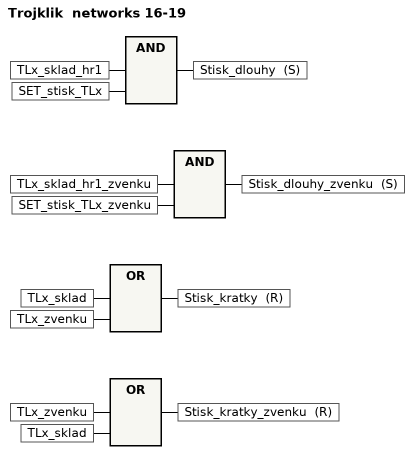
[picture p24: Trojklik (FBD) networks 16-19]
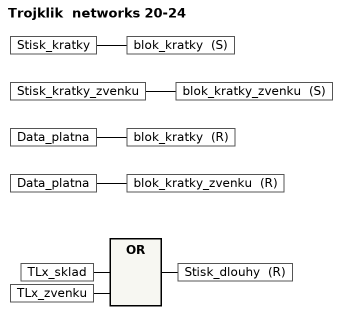
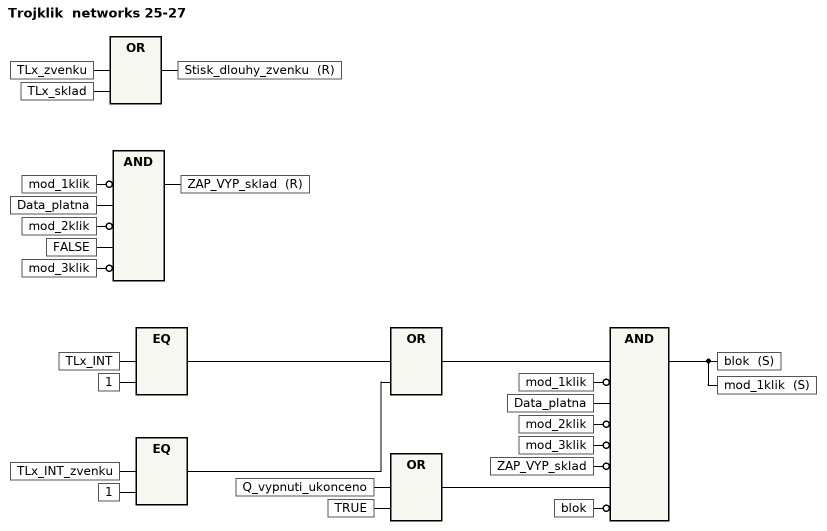
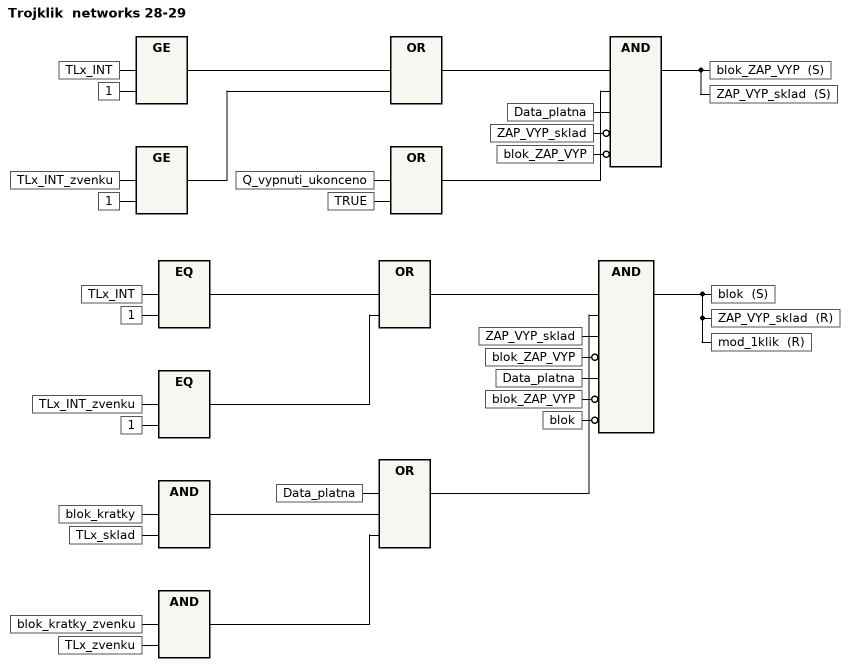
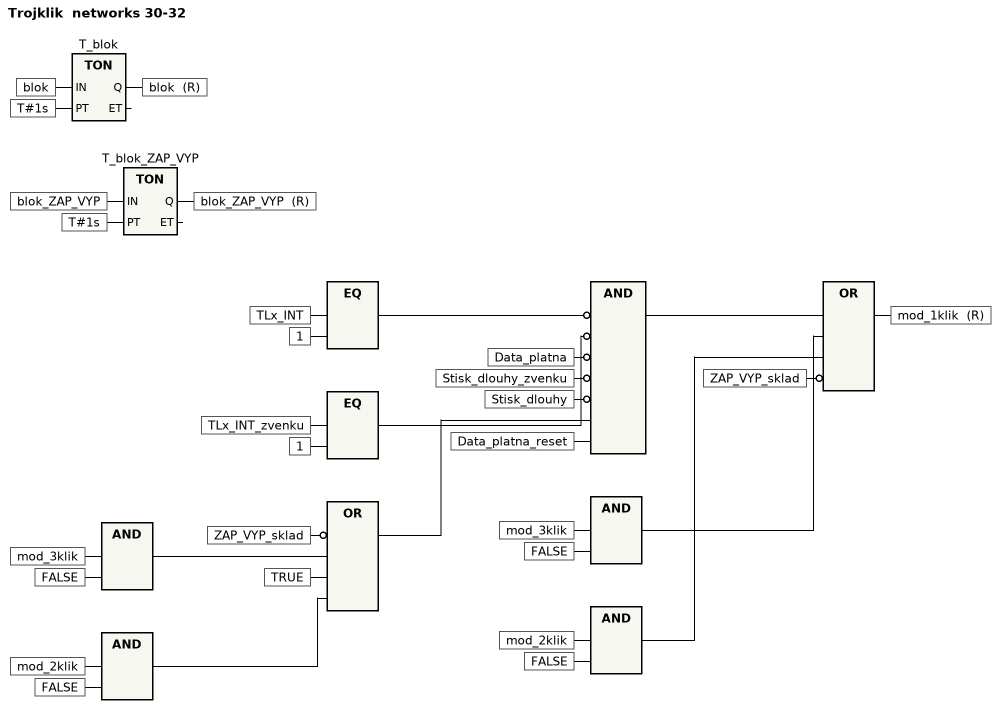
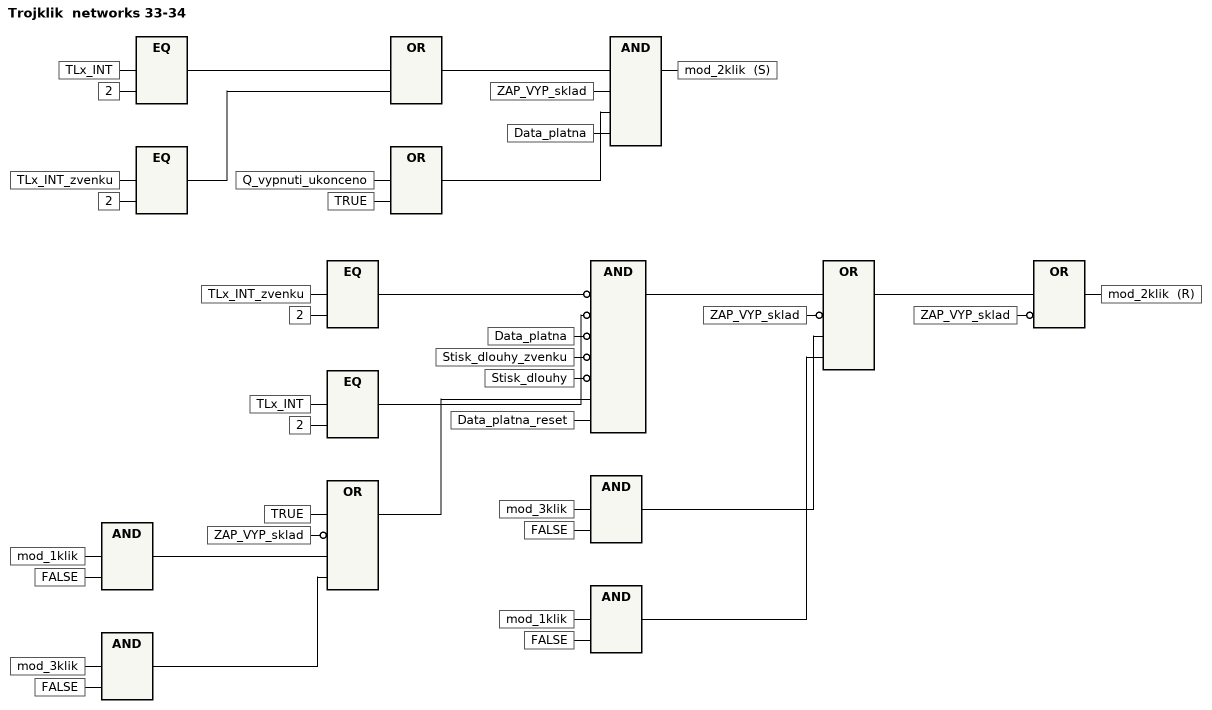
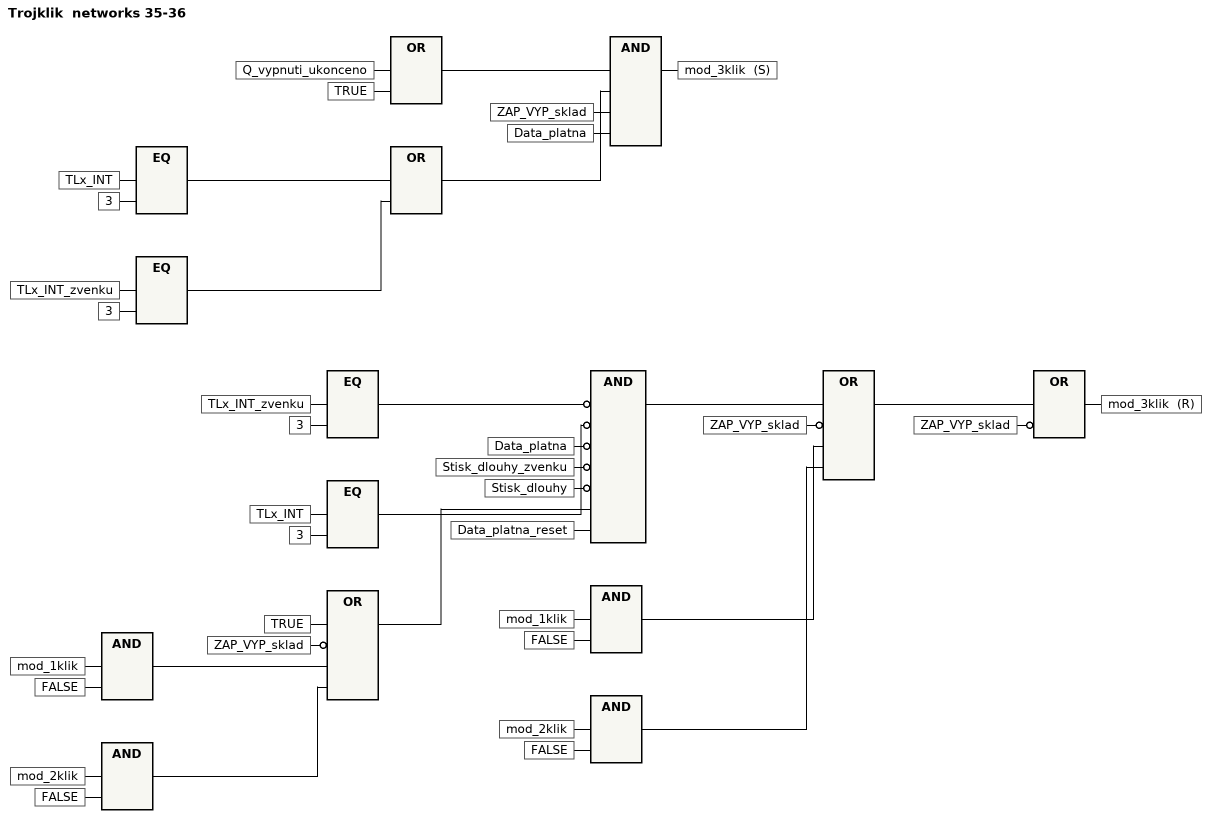
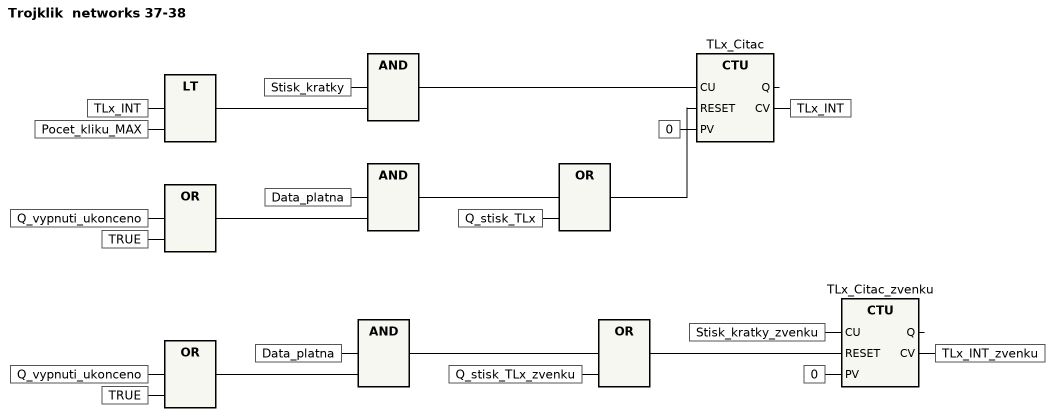
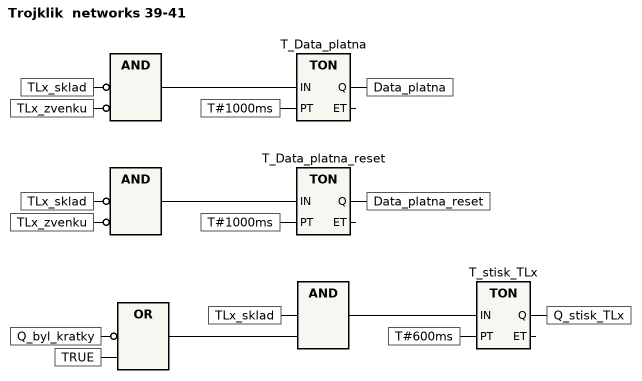
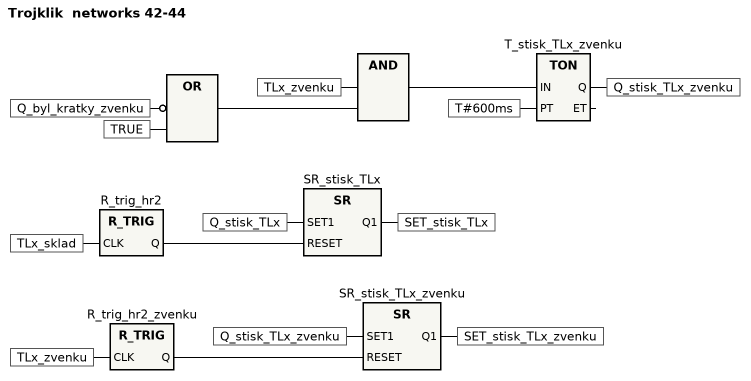
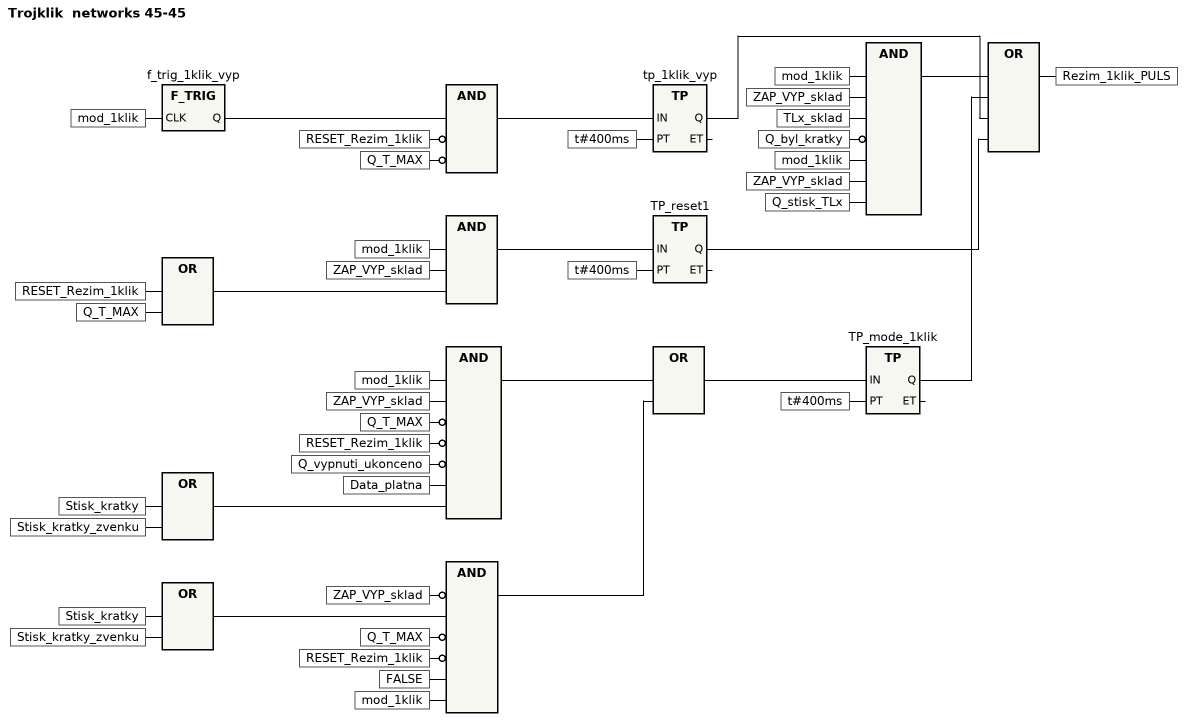
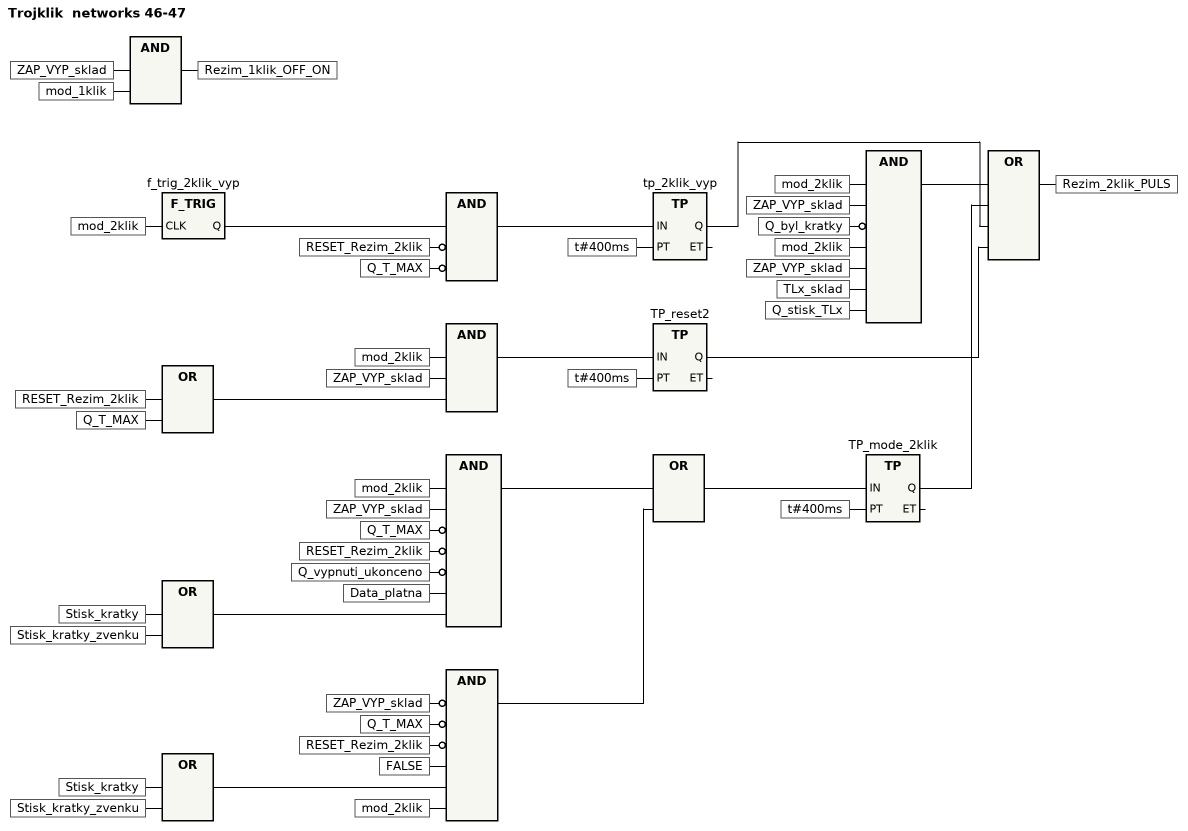
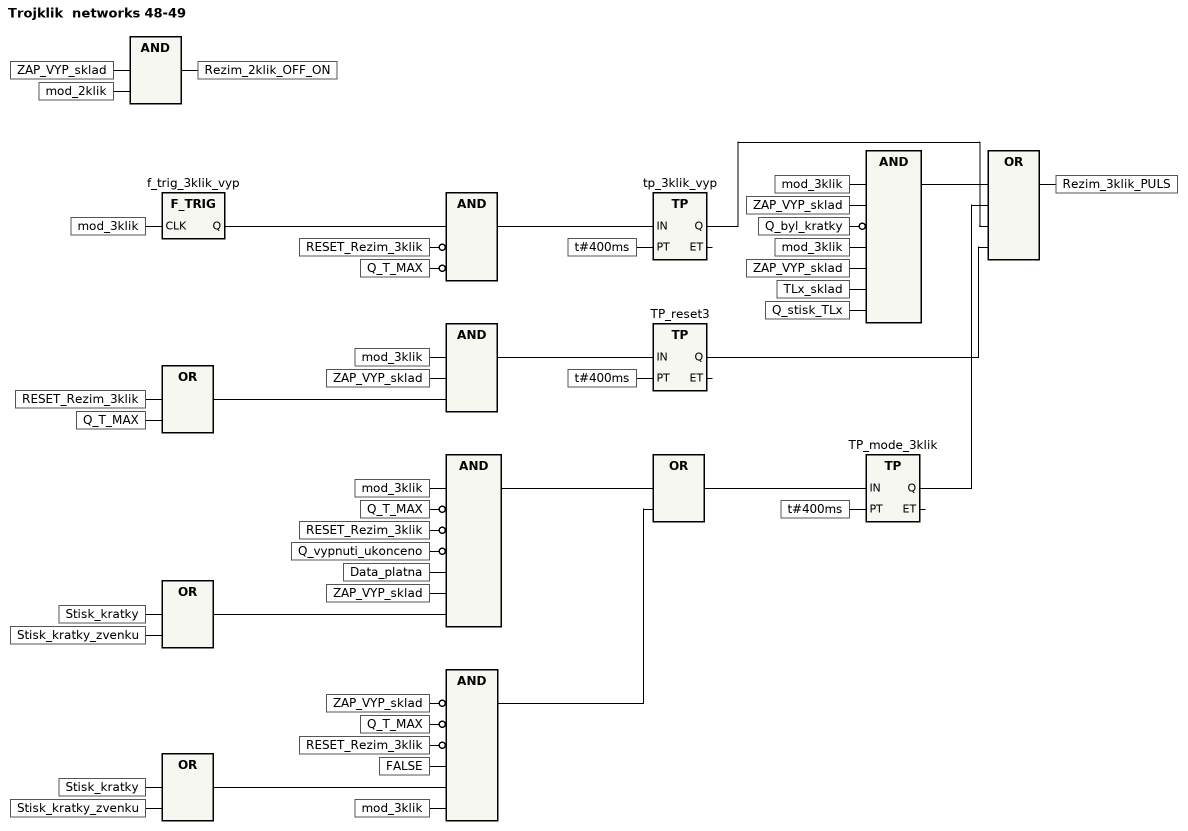
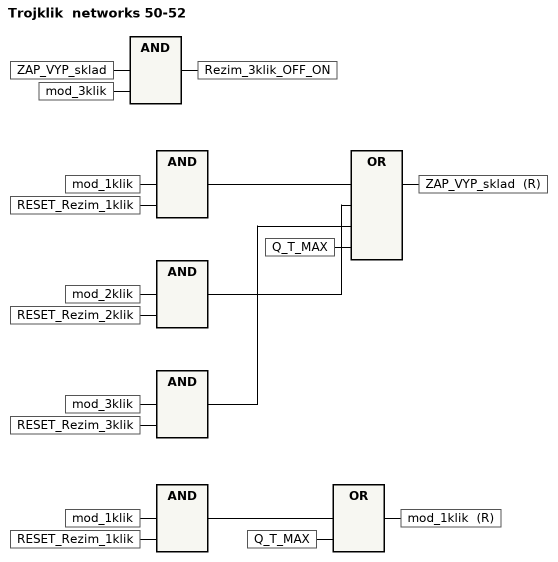
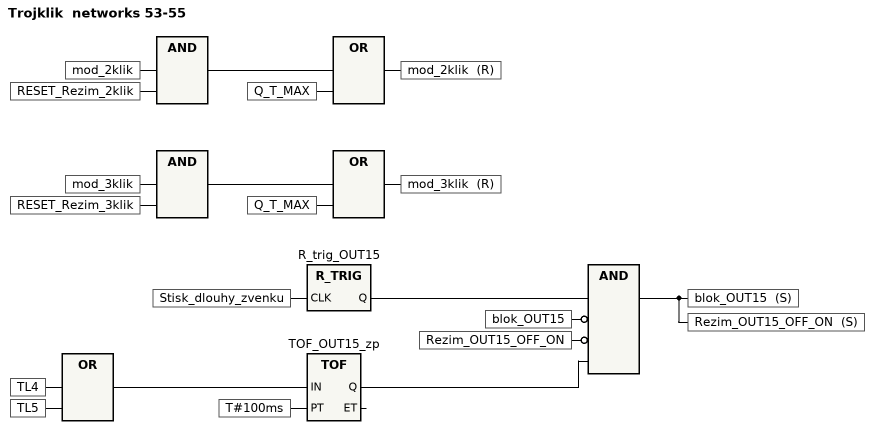
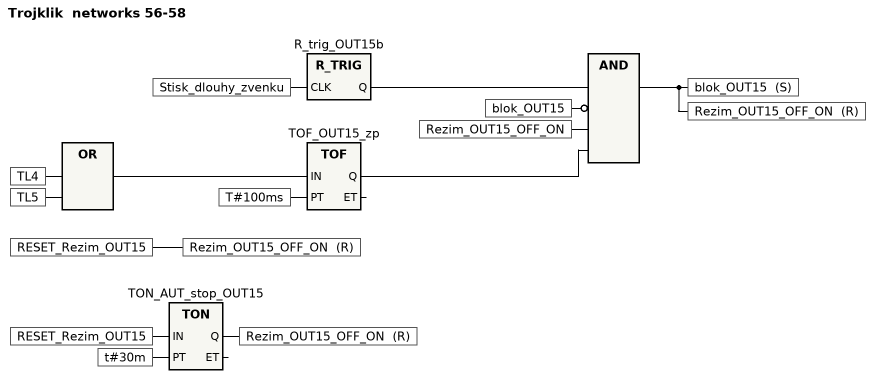
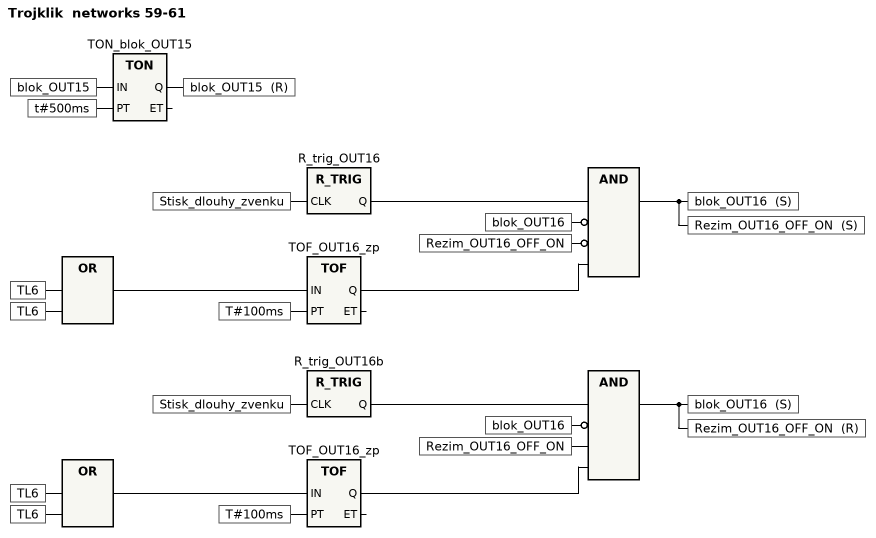
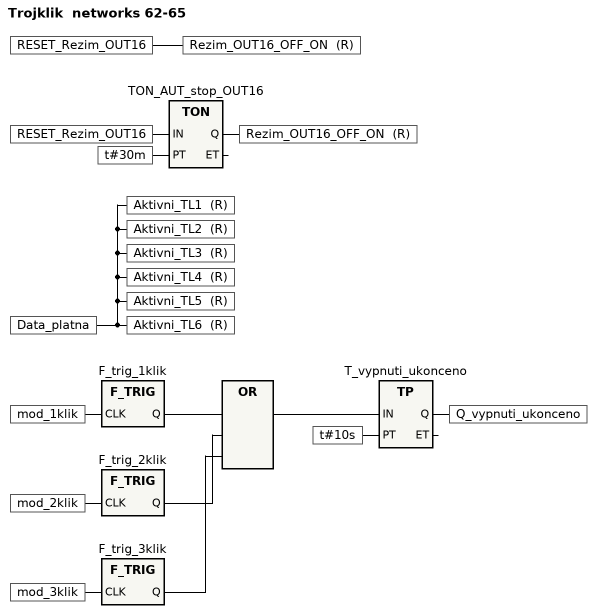
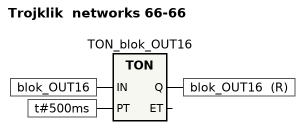
_FBD_ (* Function Block Diagram *)
NETWORK 1
	TP_T_max:TP(IN: T_max:TON(IN: AND(OR(Rezim_1klik_OFF_ON, Rezim_2klik_OFF_ON, Rezim_3klik_OFF_ON), AUT_vyp), PT: cas_vypnuti), PT: t#400ms) => Q_T_MAX
NETWORK 2
	AND(TL1, NOT Aktivni_TL1, NOT Aktivni_TL2, NOT Aktivni_TL3, NOT Aktivni_TL4, NOT Aktivni_TL5, NOT Aktivni_TL6) => S Aktivni_TL1
NETWORK 3
	AND(TL2, NOT Aktivni_TL1, NOT Aktivni_TL2, NOT Aktivni_TL3, NOT Aktivni_TL4, NOT Aktivni_TL5, NOT Aktivni_TL6) => S Aktivni_TL2
NETWORK 4
	AND(TL3, NOT Aktivni_TL1, NOT Aktivni_TL2, NOT Aktivni_TL3, NOT Aktivni_TL4, NOT Aktivni_TL5, NOT Aktivni_TL6) => S Aktivni_TL3
NETWORK 5
	AND(TL4, NOT Aktivni_TL1, NOT Aktivni_TL2, NOT Aktivni_TL3, NOT Aktivni_TL4, NOT Aktivni_TL5, NOT Aktivni_TL6) => S Aktivni_TL4
NETWORK 6
	AND(TL5, NOT Aktivni_TL1, NOT Aktivni_TL2, NOT Aktivni_TL3, NOT Aktivni_TL4, NOT Aktivni_TL5, NOT Aktivni_TL6) => S Aktivni_TL5
NETWORK 7
	AND(TL6, NOT Aktivni_TL1, NOT Aktivni_TL2, NOT Aktivni_TL3, NOT Aktivni_TL4, NOT Aktivni_TL5, NOT Aktivni_TL6) => S Aktivni_TL6
NETWORK 8
	OR(AND(TL1, Aktivni_TL1), AND(TL2, Aktivni_TL2), AND(TL3, Aktivni_TL3)) => TLx_sklad
NETWORK 9
	OR(AND(TL4, Aktivni_TL4), AND(TL5, Aktivni_TL5), AND(TL6, Aktivni_TL6)) => TLx_zvenku
NETWORK 10
	F_trig_hr1:F_TRIG(CLK: TLx_sklad) => TLx_sklad_hr1
NETWORK 11
	F_trig_hr1_zvenku:F_TRIG(CLK: TLx_zvenku) => TLx_sklad_hr1_zvenku
NETWORK 12
	AND(TLx_sklad_hr1, NOT SET_stisk_TLx) => S Stisk_kratky
NETWORK 13
	AND(TLx_sklad_hr1_zvenku, NOT SET_stisk_TLx_zvenku) => S Stisk_kratky_zvenku
NETWORK 14
	TP_byl_kratky:TP(IN: Stisk_kratky, PT: T#4s) => Q_byl_kratky
NETWORK 15
	TP_byl_kratky_zvenku:TP(IN: Stisk_kratky_zvenku, PT: T#4s) => Q_byl_kratky_zvenku
NETWORK 16
	AND(TLx_sklad_hr1, SET_stisk_TLx) => S Stisk_dlouhy
NETWORK 17
	AND(TLx_sklad_hr1_zvenku, SET_stisk_TLx_zvenku) => S Stisk_dlouhy_zvenku
NETWORK 18
	OR(TLx_sklad, TLx_zvenku) => R Stisk_kratky
NETWORK 19
	OR(TLx_zvenku, TLx_sklad) => R Stisk_kratky_zvenku
NETWORK 20
	Stisk_kratky => S blok_kratky
NETWORK 21
	Stisk_kratky_zvenku => S blok_kratky_zvenku
NETWORK 22
	Data_platna => R blok_kratky
NETWORK 23
	Data_platna => R blok_kratky_zvenku
NETWORK 24
	OR(TLx_sklad, TLx_zvenku) => R Stisk_dlouhy
NETWORK 25
	OR(TLx_zvenku, TLx_sklad) => R Stisk_dlouhy_zvenku
NETWORK 26
	AND(NOT mod_1klik, Data_platna, NOT mod_2klik, FALSE, NOT mod_3klik) => R ZAP_VYP_sklad
NETWORK 27
	AND(OR(EQ(TLx_INT, 1), EQ(TLx_INT_zvenku, 1)), NOT mod_1klik, Data_platna, NOT mod_2klik, NOT mod_3klik, NOT ZAP_VYP_sklad, OR(Q_vypnuti_ukonceno, TRUE), NOT blok) => S blok, S mod_1klik
NETWORK 28
	AND(OR(GE(TLx_INT, 1), GE(TLx_INT_zvenku, 1)), OR(Q_vypnuti_ukonceno, TRUE), Data_platna, NOT ZAP_VYP_sklad, NOT blok_ZAP_VYP) => S blok_ZAP_VYP, S ZAP_VYP_sklad
NETWORK 29
	AND(OR(EQ(TLx_INT, 1), EQ(TLx_INT_zvenku, 1)), OR(Data_platna, AND(blok_kratky, TLx_sklad), AND(blok_kratky_zvenku, TLx_zvenku)), ZAP_VYP_sklad, NOT blok_ZAP_VYP, Data_platna, NOT blok_ZAP_VYP, NOT blok) => S blok, R ZAP_VYP_sklad, R mod_1klik
NETWORK 30
	T_blok:TON(IN: blok, PT: T#1s) => R blok
NETWORK 31
	T_blok_ZAP_VYP:TON(IN: blok_ZAP_VYP, PT: T#1s) => R blok_ZAP_VYP
NETWORK 32
	OR(AND(NOT EQ(TLx_INT, 1), NOT EQ(TLx_INT_zvenku, 1), NOT Data_platna, NOT Stisk_dlouhy_zvenku, NOT Stisk_dlouhy, OR(NOT ZAP_VYP_sklad, AND(mod_3klik, FALSE), TRUE, AND(mod_2klik, FALSE)), Data_platna_reset), AND(mod_3klik, FALSE), AND(mod_2klik, FALSE), NOT ZAP_VYP_sklad) => R mod_1klik
NETWORK 33
	AND(OR(EQ(TLx_INT, 2), EQ(TLx_INT_zvenku, 2)), ZAP_VYP_sklad, OR(Q_vypnuti_ukonceno, TRUE), Data_platna) => S mod_2klik
NETWORK 34
	OR(OR(AND(NOT EQ(TLx_INT_zvenku, 2), NOT EQ(TLx_INT, 2), NOT Data_platna, NOT Stisk_dlouhy_zvenku, NOT Stisk_dlouhy, OR(TRUE, NOT ZAP_VYP_sklad, AND(mod_1klik, FALSE), AND(mod_3klik, FALSE)), Data_platna_reset), NOT ZAP_VYP_sklad, AND(mod_3klik, FALSE), AND(mod_1klik, FALSE)), NOT ZAP_VYP_sklad) => R mod_2klik
NETWORK 35
	AND(OR(Q_vypnuti_ukonceno, TRUE), OR(EQ(TLx_INT, 3), EQ(TLx_INT_zvenku, 3)), ZAP_VYP_sklad, Data_platna) => S mod_3klik
NETWORK 36
	OR(OR(AND(NOT EQ(TLx_INT_zvenku, 3), NOT EQ(TLx_INT, 3), NOT Data_platna, NOT Stisk_dlouhy_zvenku, NOT Stisk_dlouhy, OR(TRUE, NOT ZAP_VYP_sklad, AND(mod_1klik, FALSE), AND(mod_2klik, FALSE)), Data_platna_reset), NOT ZAP_VYP_sklad, AND(mod_1klik, FALSE), AND(mod_2klik, FALSE)), NOT ZAP_VYP_sklad) => R mod_3klik
NETWORK 37
	TLx_Citac:CTU(CU: AND(Stisk_kratky, LT(TLx_INT, Pocet_kliku_MAX)), RESET: OR(AND(Data_platna, OR(Q_vypnuti_ukonceno, TRUE)), Q_stisk_TLx), PV: 0, CV => TLx_INT)
NETWORK 38
	TLx_Citac_zvenku:CTU(CU: Stisk_kratky_zvenku, RESET: OR(AND(Data_platna, OR(Q_vypnuti_ukonceno, TRUE)), Q_stisk_TLx_zvenku), PV: 0, CV => TLx_INT_zvenku)
NETWORK 39 (* Data platna *)
	T_Data_platna:TON(IN: AND(NOT TLx_sklad, NOT TLx_zvenku), PT: T#1000ms) => Data_platna
NETWORK 40 (* Data platna *)
	T_Data_platna_reset:TON(IN: AND(NOT TLx_sklad, NOT TLx_zvenku), PT: T#1000ms) => Data_platna_reset
NETWORK 41 (* delka stisku TLx *)
	T_stisk_TLx:TON(IN: AND(TLx_sklad, OR(NOT Q_byl_kratky, TRUE)), PT: T#600ms) => Q_stisk_TLx
NETWORK 42 (* delka stisku TLx *)
	T_stisk_TLx_zvenku:TON(IN: AND(TLx_zvenku, OR(NOT Q_byl_kratky_zvenku, TRUE)), PT: T#600ms) => Q_stisk_TLx_zvenku
NETWORK 43
	SR_stisk_TLx:SR(SET1: Q_stisk_TLx, RESET: R_trig_hr2:R_TRIG(CLK: TLx_sklad)) => SET_stisk_TLx
NETWORK 44
	SR_stisk_TLx_zvenku:SR(SET1: Q_stisk_TLx_zvenku, RESET: R_trig_hr2_zvenku:R_TRIG(CLK: TLx_zvenku)) => SET_stisk_TLx_zvenku
NETWORK 45
	OR(AND(mod_1klik, ZAP_VYP_sklad, TLx_sklad, NOT Q_byl_kratky, mod_1klik, ZAP_VYP_sklad, Q_stisk_TLx), TP_mode_1klik:TP(IN: OR(AND(mod_1klik, ZAP_VYP_sklad, NOT Q_T_MAX, NOT RESET_Rezim_1klik, NOT Q_vypnuti_ukonceno, Data_platna, OR(Stisk_kratky, Stisk_kratky_zvenku)), AND(NOT ZAP_VYP_sklad, OR(Stisk_kratky, Stisk_kratky_zvenku), NOT Q_T_MAX, NOT RESET_Rezim_1klik, FALSE, mod_1klik)), PT: t#400ms), tp_1klik_vyp:TP(IN: AND(f_trig_1klik_vyp:F_TRIG(CLK: mod_1klik), NOT RESET_Rezim_1klik, NOT Q_T_MAX), PT: t#400ms), TP_reset1:TP(IN: AND(mod_1klik, ZAP_VYP_sklad, OR(RESET_Rezim_1klik, Q_T_MAX)), PT: t#400ms)) => Rezim_1klik_PULS
NETWORK 46
	AND(ZAP_VYP_sklad, mod_1klik) => Rezim_1klik_OFF_ON
NETWORK 47
	OR(AND(mod_2klik, ZAP_VYP_sklad, NOT Q_byl_kratky, mod_2klik, ZAP_VYP_sklad, TLx_sklad, Q_stisk_TLx), TP_mode_2klik:TP(IN: OR(AND(mod_2klik, ZAP_VYP_sklad, NOT Q_T_MAX, NOT RESET_Rezim_2klik, NOT Q_vypnuti_ukonceno, Data_platna, OR(Stisk_kratky, Stisk_kratky_zvenku)), AND(NOT ZAP_VYP_sklad, NOT Q_T_MAX, NOT RESET_Rezim_2klik, FALSE, OR(Stisk_kratky, Stisk_kratky_zvenku), mod_2klik)), PT: t#400ms), tp_2klik_vyp:TP(IN: AND(f_trig_2klik_vyp:F_TRIG(CLK: mod_2klik), NOT RESET_Rezim_2klik, NOT Q_T_MAX), PT: t#400ms), TP_reset2:TP(IN: AND(mod_2klik, ZAP_VYP_sklad, OR(RESET_Rezim_2klik, Q_T_MAX)), PT: t#400ms)) => Rezim_2klik_PULS
NETWORK 48
	AND(ZAP_VYP_sklad, mod_2klik) => Rezim_2klik_OFF_ON
NETWORK 49
	OR(AND(mod_3klik, ZAP_VYP_sklad, NOT Q_byl_kratky, mod_3klik, ZAP_VYP_sklad, TLx_sklad, Q_stisk_TLx), TP_mode_3klik:TP(IN: OR(AND(mod_3klik, NOT Q_T_MAX, NOT RESET_Rezim_3klik, NOT Q_vypnuti_ukonceno, Data_platna, ZAP_VYP_sklad, OR(Stisk_kratky, Stisk_kratky_zvenku)), AND(NOT ZAP_VYP_sklad, NOT Q_T_MAX, NOT RESET_Rezim_3klik, FALSE, OR(Stisk_kratky, Stisk_kratky_zvenku), mod_3klik)), PT: t#400ms), tp_3klik_vyp:TP(IN: AND(f_trig_3klik_vyp:F_TRIG(CLK: mod_3klik), NOT RESET_Rezim_3klik, NOT Q_T_MAX), PT: t#400ms), TP_reset3:TP(IN: AND(mod_3klik, ZAP_VYP_sklad, OR(RESET_Rezim_3klik, Q_T_MAX)), PT: t#400ms)) => Rezim_3klik_PULS
NETWORK 50
	AND(ZAP_VYP_sklad, mod_3klik) => Rezim_3klik_OFF_ON
NETWORK 51
	OR(AND(mod_1klik, RESET_Rezim_1klik), AND(mod_2klik, RESET_Rezim_2klik), AND(mod_3klik, RESET_Rezim_3klik), Q_T_MAX) => R ZAP_VYP_sklad
NETWORK 52
	OR(AND(mod_1klik, RESET_Rezim_1klik), Q_T_MAX) => R mod_1klik
NETWORK 53
	OR(AND(mod_2klik, RESET_Rezim_2klik), Q_T_MAX) => R mod_2klik
NETWORK 54
	OR(AND(mod_3klik, RESET_Rezim_3klik), Q_T_MAX) => R mod_3klik
NETWORK 55
	AND(R_trig_OUT15:R_TRIG(CLK: Stisk_dlouhy_zvenku), NOT blok_OUT15, NOT Rezim_OUT15_OFF_ON, TOF_OUT15_zp:TOF(IN: OR(TL4, TL5), PT: T#100ms)) => S blok_OUT15, S Rezim_OUT15_OFF_ON
NETWORK 56
	AND(R_trig_OUT15b:R_TRIG(CLK: Stisk_dlouhy_zvenku), NOT blok_OUT15, Rezim_OUT15_OFF_ON, TOF_OUT15_zp:TOF(IN: OR(TL4, TL5), PT: T#100ms)) => S blok_OUT15, R Rezim_OUT15_OFF_ON
NETWORK 57
	RESET_Rezim_OUT15 => R Rezim_OUT15_OFF_ON
NETWORK 58
	TON_AUT_stop_OUT15:TON(IN: RESET_Rezim_OUT15, PT: t#30m) => R Rezim_OUT15_OFF_ON
NETWORK 59
	TON_blok_OUT15:TON(IN: blok_OUT15, PT: t#500ms) => R blok_OUT15
NETWORK 60
	AND(R_trig_OUT16:R_TRIG(CLK: Stisk_dlouhy_zvenku), NOT blok_OUT16, NOT Rezim_OUT16_OFF_ON, TOF_OUT16_zp:TOF(IN: OR(TL6, TL6), PT: T#100ms)) => S blok_OUT16, S Rezim_OUT16_OFF_ON
NETWORK 61
	AND(R_trig_OUT16b:R_TRIG(CLK: Stisk_dlouhy_zvenku), NOT blok_OUT16, Rezim_OUT16_OFF_ON, TOF_OUT16_zp:TOF(IN: OR(TL6, TL6), PT: T#100ms)) => S blok_OUT16, R Rezim_OUT16_OFF_ON
NETWORK 62
	RESET_Rezim_OUT16 => R Rezim_OUT16_OFF_ON
NETWORK 63
	TON_AUT_stop_OUT16:TON(IN: RESET_Rezim_OUT16, PT: t#30m) => R Rezim_OUT16_OFF_ON
NETWORK 64
	Data_platna => R Aktivni_TL1, R Aktivni_TL2, R Aktivni_TL3, R Aktivni_TL4, R Aktivni_TL5, R Aktivni_TL6
NETWORK 65
	T_vypnuti_ukonceno:TP(IN: OR(F_trig_1klik:F_TRIG(CLK: mod_1klik), F_trig_2klik:F_TRIG(CLK: mod_2klik), F_trig_3klik:F_TRIG(CLK: mod_3klik)), PT: t#10s) => Q_vypnuti_ukonceno
NETWORK 66
	TON_blok_OUT16:TON(IN: blok_OUT16, PT: t#500ms) => R blok_OUT16
_END_FBD_
(* the same logic as Structured Text *)
(* Network 1 *)
T_max(IN := (Rezim_1klik_OFF_ON OR Rezim_2klik_OFF_ON OR Rezim_3klik_OFF_ON) AND AUT_vyp, PT := cas_vypnuti);
TP_T_max(IN := T_max.Q, PT := t#400ms);
Q_T_MAX := TP_T_max.Q;
(* Network 2 *)
IF TL1 AND NOT Aktivni_TL1 AND NOT Aktivni_TL2 AND NOT Aktivni_TL3 AND NOT Aktivni_TL4 AND NOT Aktivni_TL5 AND NOT Aktivni_TL6 THEN Aktivni_TL1 := TRUE; END_IF;
(* Network 3 *)
IF TL2 AND NOT Aktivni_TL1 AND NOT Aktivni_TL2 AND NOT Aktivni_TL3 AND NOT Aktivni_TL4 AND NOT Aktivni_TL5 AND NOT Aktivni_TL6 THEN Aktivni_TL2 := TRUE; END_IF;
(* Network 4 *)
IF TL3 AND NOT Aktivni_TL1 AND NOT Aktivni_TL2 AND NOT Aktivni_TL3 AND NOT Aktivni_TL4 AND NOT Aktivni_TL5 AND NOT Aktivni_TL6 THEN Aktivni_TL3 := TRUE; END_IF;
(* Network 5 *)
IF TL4 AND NOT Aktivni_TL1 AND NOT Aktivni_TL2 AND NOT Aktivni_TL3 AND NOT Aktivni_TL4 AND NOT Aktivni_TL5 AND NOT Aktivni_TL6 THEN Aktivni_TL4 := TRUE; END_IF;
(* Network 6 *)
IF TL5 AND NOT Aktivni_TL1 AND NOT Aktivni_TL2 AND NOT Aktivni_TL3 AND NOT Aktivni_TL4 AND NOT Aktivni_TL5 AND NOT Aktivni_TL6 THEN Aktivni_TL5 := TRUE; END_IF;
(* Network 7 *)
IF TL6 AND NOT Aktivni_TL1 AND NOT Aktivni_TL2 AND NOT Aktivni_TL3 AND NOT Aktivni_TL4 AND NOT Aktivni_TL5 AND NOT Aktivni_TL6 THEN Aktivni_TL6 := TRUE; END_IF;
(* Network 8 *)
TLx_sklad := (TL1 AND Aktivni_TL1) OR (TL2 AND Aktivni_TL2) OR (TL3 AND Aktivni_TL3);
(* Network 9 *)
TLx_zvenku := (TL4 AND Aktivni_TL4) OR (TL5 AND Aktivni_TL5) OR (TL6 AND Aktivni_TL6);
(* Network 10 *)
F_trig_hr1(CLK := TLx_sklad);
TLx_sklad_hr1 := F_trig_hr1.Q;
(* Network 11 *)
F_trig_hr1_zvenku(CLK := TLx_zvenku);
TLx_sklad_hr1_zvenku := F_trig_hr1_zvenku.Q;
(* Network 12 *)
IF TLx_sklad_hr1 AND NOT SET_stisk_TLx THEN Stisk_kratky := TRUE; END_IF;
(* Network 13 *)
IF TLx_sklad_hr1_zvenku AND NOT SET_stisk_TLx_zvenku THEN Stisk_kratky_zvenku := TRUE; END_IF;
(* Network 14 *)
TP_byl_kratky(IN := Stisk_kratky, PT := T#4s);
Q_byl_kratky := TP_byl_kratky.Q;
(* Network 15 *)
TP_byl_kratky_zvenku(IN := Stisk_kratky_zvenku, PT := T#4s);
Q_byl_kratky_zvenku := TP_byl_kratky_zvenku.Q;
(* Network 16 *)
IF TLx_sklad_hr1 AND SET_stisk_TLx THEN Stisk_dlouhy := TRUE; END_IF;
(* Network 17 *)
IF TLx_sklad_hr1_zvenku AND SET_stisk_TLx_zvenku THEN Stisk_dlouhy_zvenku := TRUE; END_IF;
(* Network 18 *)
IF TLx_sklad OR TLx_zvenku THEN Stisk_kratky := FALSE; END_IF;
(* Network 19 *)
IF TLx_zvenku OR TLx_sklad THEN Stisk_kratky_zvenku := FALSE; END_IF;
(* Network 20 *)
IF Stisk_kratky THEN blok_kratky := TRUE; END_IF;
(* Network 21 *)
IF Stisk_kratky_zvenku THEN blok_kratky_zvenku := TRUE; END_IF;
(* Network 22 *)
IF Data_platna THEN blok_kratky := FALSE; END_IF;
(* Network 23 *)
IF Data_platna THEN blok_kratky_zvenku := FALSE; END_IF;
(* Network 24 *)
IF TLx_sklad OR TLx_zvenku THEN Stisk_dlouhy := FALSE; END_IF;
(* Network 25 *)
IF TLx_zvenku OR TLx_sklad THEN Stisk_dlouhy_zvenku := FALSE; END_IF;
(* Network 26 *)
IF NOT mod_1klik AND Data_platna AND NOT mod_2klik AND FALSE AND NOT mod_3klik THEN ZAP_VYP_sklad := FALSE; END_IF;
(* Network 27 *)
_p1 := ((TLx_INT = 1) OR (TLx_INT_zvenku = 1)) AND NOT mod_1klik AND Data_platna AND NOT mod_2klik AND NOT mod_3klik AND NOT ZAP_VYP_sklad AND (Q_vypnuti_ukonceno OR TRUE) AND NOT blok;
IF _p1 THEN blok := TRUE; mod_1klik := TRUE; END_IF;
(* Network 28 *)
_p2 := ((TLx_INT >= 1) OR (TLx_INT_zvenku >= 1)) AND (Q_vypnuti_ukonceno OR TRUE) AND Data_platna AND NOT ZAP_VYP_sklad AND NOT blok_ZAP_VYP;
IF _p2 THEN blok_ZAP_VYP := TRUE; ZAP_VYP_sklad := TRUE; END_IF;
(* Network 29 *)
_p3 := ((TLx_INT = 1) OR (TLx_INT_zvenku = 1)) AND (Data_platna OR (blok_kratky AND TLx_sklad) OR (blok_kratky_zvenku AND TLx_zvenku)) AND ZAP_VYP_sklad AND NOT blok_ZAP_VYP AND Data_platna AND NOT blok_ZAP_VYP AND NOT blok;
IF _p3 THEN blok := TRUE; ZAP_VYP_sklad := FALSE; mod_1klik := FALSE; END_IF;
(* Network 30 *)
T_blok(IN := blok, PT := T#1s);
IF T_blok.Q THEN blok := FALSE; END_IF;
(* Network 31 *)
T_blok_ZAP_VYP(IN := blok_ZAP_VYP, PT := T#1s);
IF T_blok_ZAP_VYP.Q THEN blok_ZAP_VYP := FALSE; END_IF;
(* Network 32 *)
IF (NOT (TLx_INT = 1) AND NOT (TLx_INT_zvenku = 1) AND NOT Data_platna AND NOT Stisk_dlouhy_zvenku AND NOT Stisk_dlouhy AND (NOT ZAP_VYP_sklad OR (mod_3klik AND FALSE) OR TRUE OR (mod_2klik AND FALSE)) AND Data_platna_reset) OR (mod_3klik AND FALSE) OR (mod_2klik AND FALSE) OR NOT ZAP_VYP_sklad THEN mod_1klik := FALSE; END_IF;
(* Network 33 *)
IF ((TLx_INT = 2) OR (TLx_INT_zvenku = 2)) AND ZAP_VYP_sklad AND (Q_vypnuti_ukonceno OR TRUE) AND Data_platna THEN mod_2klik := TRUE; END_IF;
(* Network 34 *)
IF ((NOT (TLx_INT_zvenku = 2) AND NOT (TLx_INT = 2) AND NOT Data_platna AND NOT Stisk_dlouhy_zvenku AND NOT Stisk_dlouhy AND (TRUE OR NOT ZAP_VYP_sklad OR (mod_1klik AND FALSE) OR (mod_3klik AND FALSE)) AND Data_platna_reset) OR NOT ZAP_VYP_sklad OR (mod_3klik AND FALSE) OR (mod_1klik AND FALSE)) OR NOT ZAP_VYP_sklad THEN mod_2klik := FALSE; END_IF;
(* Network 35 *)
IF (Q_vypnuti_ukonceno OR TRUE) AND ((TLx_INT = 3) OR (TLx_INT_zvenku = 3)) AND ZAP_VYP_sklad AND Data_platna THEN mod_3klik := TRUE; END_IF;
(* Network 36 *)
IF ((NOT (TLx_INT_zvenku = 3) AND NOT (TLx_INT = 3) AND NOT Data_platna AND NOT Stisk_dlouhy_zvenku AND NOT Stisk_dlouhy AND (TRUE OR NOT ZAP_VYP_sklad OR (mod_1klik AND FALSE) OR (mod_2klik AND FALSE)) AND Data_platna_reset) OR NOT ZAP_VYP_sklad OR (mod_1klik AND FALSE) OR (mod_2klik AND FALSE)) OR NOT ZAP_VYP_sklad THEN mod_3klik := FALSE; END_IF;
(* Network 37 *)
TLx_Citac(CU := Stisk_kratky AND (TLx_INT < Pocet_kliku_MAX), RESET := (Data_platna AND (Q_vypnuti_ukonceno OR TRUE)) OR Q_stisk_TLx, PV := 0);
TLx_INT := TLx_Citac.CV;
(* Network 38 *)
TLx_Citac_zvenku(CU := Stisk_kratky_zvenku, RESET := (Data_platna AND (Q_vypnuti_ukonceno OR TRUE)) OR Q_stisk_TLx_zvenku, PV := 0);
TLx_INT_zvenku := TLx_Citac_zvenku.CV;
(* Network 39 *)
T_Data_platna(IN := NOT TLx_sklad AND NOT TLx_zvenku, PT := T#1000ms);
Data_platna := T_Data_platna.Q;
(* Network 40 *)
T_Data_platna_reset(IN := NOT TLx_sklad AND NOT TLx_zvenku, PT := T#1000ms);
Data_platna_reset := T_Data_platna_reset.Q;
(* Network 41: see the listing above *)
(* Network 42: see the listing above *)
(* Network 43 *)
R_trig_hr2(CLK := TLx_sklad);
SR_stisk_TLx(SET1 := Q_stisk_TLx, RESET := R_trig_hr2.Q);
SET_stisk_TLx := SR_stisk_TLx.Q1;
(* Network 44 *)
R_trig_hr2_zvenku(CLK := TLx_zvenku);
SR_stisk_TLx_zvenku(SET1 := Q_stisk_TLx_zvenku, RESET := R_trig_hr2_zvenku.Q);
SET_stisk_TLx_zvenku := SR_stisk_TLx_zvenku.Q1;
(* Network 45 *)
TP_mode_1klik(IN := (mod_1klik AND ZAP_VYP_sklad AND NOT Q_T_MAX AND NOT RESET_Rezim_1klik AND NOT Q_vypnuti_ukonceno AND Data_platna AND (Stisk_kratky OR Stisk_kratky_zvenku)) OR (NOT ZAP_VYP_sklad AND (Stisk_kratky OR Stisk_kratky_zvenku) AND NOT Q_T_MAX AND NOT RESET_Rezim_1klik AND FALSE AND mod_1klik), PT := t#400ms);
f_trig_1klik_vyp(CLK := mod_1klik);
tp_1klik_vyp(IN := f_trig_1klik_vyp.Q AND NOT RESET_Rezim_1klik AND NOT Q_T_MAX, PT := t#400ms);
TP_reset1(IN := mod_1klik AND ZAP_VYP_sklad AND (RESET_Rezim_1klik OR Q_T_MAX), PT := t#400ms);
Rezim_1klik_PULS := (mod_1klik AND ZAP_VYP_sklad AND TLx_sklad AND NOT Q_byl_kratky AND mod_1klik AND ZAP_VYP_sklad AND Q_stisk_TLx) OR TP_mode_1klik.Q OR tp_1klik_vyp.Q OR TP_reset1.Q;
(* Network 46 *)
Rezim_1klik_OFF_ON := ZAP_VYP_sklad AND mod_1klik;
(* Network 47 *)
TP_mode_2klik(IN := (mod_2klik AND ZAP_VYP_sklad AND NOT Q_T_MAX AND NOT RESET_Rezim_2klik AND NOT Q_vypnuti_ukonceno AND Data_platna AND (Stisk_kratky OR Stisk_kratky_zvenku)) OR (NOT ZAP_VYP_sklad AND NOT Q_T_MAX AND NOT RESET_Rezim_2klik AND FALSE AND (Stisk_kratky OR Stisk_kratky_zvenku) AND mod_2klik), PT := t#400ms);
f_trig_2klik_vyp(CLK := mod_2klik);
tp_2klik_vyp(IN := f_trig_2klik_vyp.Q AND NOT RESET_Rezim_2klik AND NOT Q_T_MAX, PT := t#400ms);
TP_reset2(IN := mod_2klik AND ZAP_VYP_sklad AND (RESET_Rezim_2klik OR Q_T_MAX), PT := t#400ms);
Rezim_2klik_PULS := (mod_2klik AND ZAP_VYP_sklad AND NOT Q_byl_kratky AND mod_2klik AND ZAP_VYP_sklad AND TLx_sklad AND Q_stisk_TLx) OR TP_mode_2klik.Q OR tp_2klik_vyp.Q OR TP_reset2.Q;
(* Network 48 *)
Rezim_2klik_OFF_ON := ZAP_VYP_sklad AND mod_2klik;
(* Network 49 *)
TP_mode_3klik(IN := (mod_3klik AND NOT Q_T_MAX AND NOT RESET_Rezim_3klik AND NOT Q_vypnuti_ukonceno AND Data_platna AND ZAP_VYP_sklad AND (Stisk_kratky OR Stisk_kratky_zvenku)) OR (NOT ZAP_VYP_sklad AND NOT Q_T_MAX AND NOT RESET_Rezim_3klik AND FALSE AND (Stisk_kratky OR Stisk_kratky_zvenku) AND mod_3klik), PT := t#400ms);
f_trig_3klik_vyp(CLK := mod_3klik);
tp_3klik_vyp(IN := f_trig_3klik_vyp.Q AND NOT RESET_Rezim_3klik AND NOT Q_T_MAX, PT := t#400ms);
TP_reset3(IN := mod_3klik AND ZAP_VYP_sklad AND (RESET_Rezim_3klik OR Q_T_MAX), PT := t#400ms);
Rezim_3klik_PULS := (mod_3klik AND ZAP_VYP_sklad AND NOT Q_byl_kratky AND mod_3klik AND ZAP_VYP_sklad AND TLx_sklad AND Q_stisk_TLx) OR TP_mode_3klik.Q OR tp_3klik_vyp.Q OR TP_reset3.Q;
(* Network 50 *)
Rezim_3klik_OFF_ON := ZAP_VYP_sklad AND mod_3klik;
(* Network 51 *)
IF (mod_1klik AND RESET_Rezim_1klik) OR (mod_2klik AND RESET_Rezim_2klik) OR (mod_3klik AND RESET_Rezim_3klik) OR Q_T_MAX THEN ZAP_VYP_sklad := FALSE; END_IF;
(* Network 52 *)
IF (mod_1klik AND RESET_Rezim_1klik) OR Q_T_MAX THEN mod_1klik := FALSE; END_IF;
(* Network 53 *)
IF (mod_2klik AND RESET_Rezim_2klik) OR Q_T_MAX THEN mod_2klik := FALSE; END_IF;
(* Network 54 *)
IF (mod_3klik AND RESET_Rezim_3klik) OR Q_T_MAX THEN mod_3klik := FALSE; END_IF;
(* Network 55 *)
R_trig_OUT15(CLK := Stisk_dlouhy_zvenku);
TOF_OUT15_zp(IN := TL4 OR TL5, PT := T#100ms);
_p4 := R_trig_OUT15.Q AND NOT blok_OUT15 AND NOT Rezim_OUT15_OFF_ON AND TOF_OUT15_zp.Q;
IF _p4 THEN blok_OUT15 := TRUE; Rezim_OUT15_OFF_ON := TRUE; END_IF;
(* Network 56 *)
R_trig_OUT15b(CLK := Stisk_dlouhy_zvenku);
TOF_OUT15_zp(IN := TL4 OR TL5, PT := T#100ms);
_p5 := R_trig_OUT15b.Q AND NOT blok_OUT15 AND Rezim_OUT15_OFF_ON AND TOF_OUT15_zp.Q;
IF _p5 THEN blok_OUT15 := TRUE; Rezim_OUT15_OFF_ON := FALSE; END_IF;
(* Network 57 *)
IF RESET_Rezim_OUT15 THEN Rezim_OUT15_OFF_ON := FALSE; END_IF;
(* Network 58 *)
TON_AUT_stop_OUT15(IN := RESET_Rezim_OUT15, PT := t#30m);
IF TON_AUT_stop_OUT15.Q THEN Rezim_OUT15_OFF_ON := FALSE; END_IF;
(* Network 59 *)
TON_blok_OUT15(IN := blok_OUT15, PT := t#500ms);
IF TON_blok_OUT15.Q THEN blok_OUT15 := FALSE; END_IF;
(* Network 60 *)
R_trig_OUT16(CLK := Stisk_dlouhy_zvenku);
TOF_OUT16_zp(IN := TL6 OR TL6, PT := T#100ms);
_p6 := R_trig_OUT16.Q AND NOT blok_OUT16 AND NOT Rezim_OUT16_OFF_ON AND TOF_OUT16_zp.Q;
IF _p6 THEN blok_OUT16 := TRUE; Rezim_OUT16_OFF_ON := TRUE; END_IF;
(* Network 61 *)
R_trig_OUT16b(CLK := Stisk_dlouhy_zvenku);
TOF_OUT16_zp(IN := TL6 OR TL6, PT := T#100ms);
_p7 := R_trig_OUT16b.Q AND NOT blok_OUT16 AND Rezim_OUT16_OFF_ON AND TOF_OUT16_zp.Q;
IF _p7 THEN blok_OUT16 := TRUE; Rezim_OUT16_OFF_ON := FALSE; END_IF;
(* Network 62 *)
IF RESET_Rezim_OUT16 THEN Rezim_OUT16_OFF_ON := FALSE; END_IF;
(* Network 63 *)
TON_AUT_stop_OUT16(IN := RESET_Rezim_OUT16, PT := t#30m);
IF TON_AUT_stop_OUT16.Q THEN Rezim_OUT16_OFF_ON := FALSE; END_IF;
(* Network 64 *)
IF Data_platna THEN Aktivni_TL1 := FALSE; Aktivni_TL2 := FALSE; Aktivni_TL3 := FALSE; Aktivni_TL4 := FALSE; Aktivni_TL5 := FALSE; Aktivni_TL6 := FALSE; END_IF;
(* Network 65 *)
F_trig_1klik(CLK := mod_1klik);
F_trig_2klik(CLK := mod_2klik);
F_trig_3klik(CLK := mod_3klik);
T_vypnuti_ukonceno(IN := F_trig_1klik.Q OR F_trig_2klik.Q OR F_trig_3klik.Q, PT := t#10s);
Q_vypnuti_ukonceno := T_vypnuti_ukonceno.Q;
(* Network 66 *)
TON_blok_OUT16(IN := blok_OUT16, PT := t#500ms);
IF TON_blok_OUT16.Q THEN blok_OUT16 := FALSE; END_IF;
END_FUNCTION_BLOCK

(* POU Zhasni, ST *)
FUNCTION_BLOCK Zhasni
VAR_INPUT
	wIn: WORD;
	xPresun: BOOL;
END_VAR
VAR_OUTPUT
	xonOUT1: BOOL;
	xonOUT2: BOOL;
	xonOUT3: BOOL;

	xoffOUT1: BOOL;
	xoffOUT2: BOOL;
	xoffOUT3: BOOL;
	wLast: WORD;
	xPresunuto: BOOL;
END_VAR
VAR
	start: BOOL;
	TP1: TP;
	stav: WORD;
	last: WORD;
	F_TRIG5: F_TRIG;
END_VAR
IF xPresun=TRUE THEN
	stav:=wIn;
	start:=TRUE;


CASE stav OF
	2: 	xonOUT2:=TRUE;
		last:=2;
	3: 	xonOUT3:=TRUE;
		last:=3;
END_CASE


IF wLast=0 AND stav=1 THEN
xonOUT1:=TRUE;
last:=1;
END_IF

IF NOT( wLast=0) AND stav=1 THEN
	CASE wLast OF
	1: xoffOUT1:=TRUE;
		last:=0;
	2: xoffOUT2:=TRUE;
		last:=0;
	3: xoffOUT3:=TRUE;
		last:=0;
	END_CASE

END_IF
END_IF

TP1(IN:=start , PT:=t#50ms , Q=> , ET=> );
F_TRIG5(CLK:=TP1.Q , Q=> );
IF F_TRIG5.Q=TRUE THEN
	wLast:=last;
	start:=FALSE;
	xoffOUT1:=FALSE;
	xoffOUT2:=FALSE;
	xoffOUT3:=FALSE;
	xonOUT1:=FALSE;
	xonOUT2:=FALSE;
	xonOUT3:=FALSE;
END_IF

xPresunuto:=xPresun;
END_FUNCTION_BLOCK

(* POU start, FBD *)
PROGRAM start
VAR
END_VAR
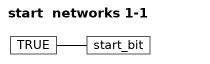
_FBD_ (* Function Block Diagram *)
NETWORK 1
	TRUE => start_bit
_END_FBD_
(* the same logic as Structured Text *)
(* Network 1 *)
start_bit := TRUE;
END_PROGRAM

(* POU TriFaze, ST *)
PROGRAM TriFaze
VAR

	Fb750_493_Master3Phase1: Fb750_493_Master3Phase;
	abIn AT %IB22: ARRAY [0..11] OF BYTE;
	abOut AT %QB6: ARRAY [0..11] OF BYTE;

	typ3faze: typConfig3Phase;
	awProud: ARRAY [1..3] OF WORD;
	awNapeti: ARRAY [1..3] OF WORD;
	aiCosFi: ARRAY [1..3] OF INT;
	aiVykon: ARRAY [1..3] OF INT;
	adwSpotreba: ARRAY [1..3] OF DWORD;

	arProud: ARRAY [1..3] OF REAL;
	arNapeti: ARRAY [1..3] OF REAL;
	arCosFi: ARRAY [1..3] OF REAL;
	arVykon: ARRAY [1..3] OF REAL;
	arSpotreba: ARRAY [1..3] OF REAL;
	SmazL1: BOOL;
	SmazL2: BOOL;
	SmazL3: BOOL;
END_VAR
Fb750_493_Master3Phase1(
	xEnable:= TRUE,
	tCycleTime:= ,
	x750_493_000_001:=FALSE ,
	xSaveEnergyConsumption:= ,
	xDeleteEnergyConsumptionL1:=SmazL1 ,
	xDeleteEnergyConsumptionL2:=SmazL1 ,
	xDeleteEnergyConsumptionL3:=SmazL1 ,
	abIn_Data_750_493:=abIn ,
	abOut_Data_750_493:=abOut ,
	typConfig3Phase:=typ3faze ,
	xReady=> ,
	abError=> , 
	awCurrent=>awProud ,
	awVoltage=>awNapeti ,
	aiPowerFactor=>aiCosFi ,
	aiEffectivePower=>aiVykon ,
	adwEnergyConsumption=>adwSpotreba ,
	awMaxCurrent=> , 
	awMaxVoltage=> , 
	awMinCurrent=> ,
	awMinVoltage=> );

arProud[1]:=awProud[1]/1000.0;
arProud[2]:=awProud[2]/1000.0;
arProud[3]:=awProud[3]/1000.0;

arNapeti[1]:=awNapeti[1]/10.0;
arNapeti[2]:=awNapeti[2]/10.0;
arNapeti[3]:=awNapeti[3]/10.0;

arCosFi[1]:=aiCosFi[1]/100.0;
arCosFi[2]:=aiCosFi[2]/100.0;
arCosFi[3]:=aiCosFi[3]/100.0;

arVykon[1]:=aiVykon[1]/10000.0;
arVykon[2]:=aiVykon[2]/10000.0;
arVykon[3]:=aiVykon[3]/10000.0;
;
END_PROGRAM

(* Visualisation Addressing
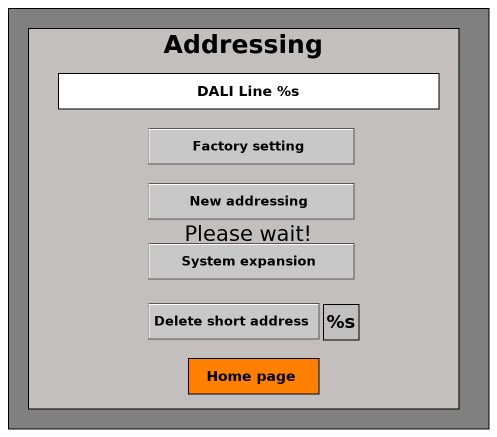
rectangle at (185,80)-(616,461): text "Addressing"
button at (305,235)-(511,271): text "New addressing"; taps DALI_Config.NewAddress; tooltip You have to click and hold the button "New Addressing" longer than two seconds to start the new addressing.
button at (305,295)-(511,331): text "System expansion"; taps DALI_Config.xErweitert; tooltip If you click the button "System expansion", only the ECGs with no short address will be addressed.
rectangle at (480,356)-(516,392): text "%s"; shows DALI_Config.LoeschKurzadr; tooltip Enter the short address to be deleted (1 - 64).; editable
rounded rectangle at (345,410)-(476,446): text "Home page"; opens DALI; tooltip Back to home page
button at (305,180)-(511,216): text "Factory setting"; taps DALI_Config.Reset; tooltip To reset the ECG you have to click and hold the button two seconds. Group and scene configurations will be deleted.
button at (305,355)-(476,391): text "Delete short address"; taps DALI_Config.Loeschen; tooltip The selected short address will be deleted.
rectangle at (265,100)-(546,471): text "Please wait!"; invisible if not DALI_Config.JobMerker[5]
rounded rectangle at (215,125)-(596,161): text "DALI Line %s"; shows DALI_Config.bDali_Linie; tooltip You can change the DALI Line only on the home page.
1 more shapes without text or variables
*)

(* Visualisation DALI
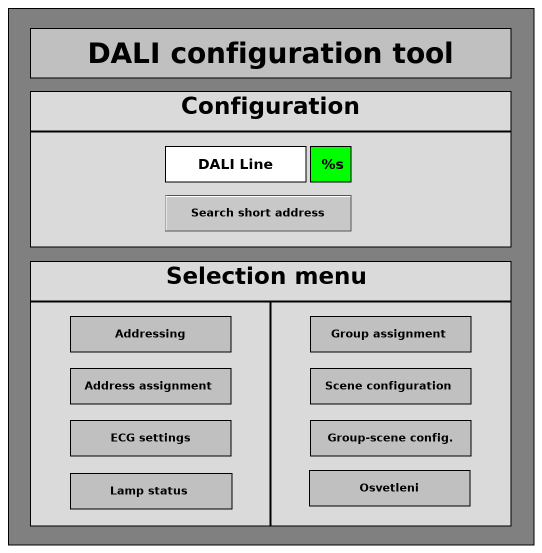
rectangle at (171,91)-(652,247): text "Configuration"
rectangle at (171,261)-(652,526): text "Selection menu"
rectangle at (171,28)-(652,78): text "DALI configuration tool"
rectangle at (211,316)-(372,352): text "Addressing"; opens Addressing
rectangle at (211,368)-(372,404): text "Address assignment"; opens Sort_short_address
rectangle at (451,316)-(612,352): text "Group assignment"; opens group_assignment
rectangle at (451,368)-(612,404): text "Scene configuration"; opens Scene_configuration
rectangle at (211,420)-(372,456): text "ECG settings"; opens ECG_settings
rectangle at (451,420)-(612,456): text "Group-scene config."; opens GroupSceneConfiguration
rectangle at (306,146)-(447,182): text "DALI Line"
button at (306,195)-(492,231): text "Search short address"; taps DALI_Config.SucheKurzadr; tooltip Clicking the button "Search Short Address" will start the search for available short addresses.
rectangle at (451,146)-(492,182): text "%s"; shows DALI_Config.Dali_Linie; alarm colour if DALI_Config.keineJobliste; tooltip Select DALI Line (1 - 5); editable
rectangle at (211,473)-(373,509): text "Lamp status"; opens Lamp_status
rectangle at (450,470)-(611,506): text "Osvetleni"; opens PLC_VISU
4 more shapes without text or variables
*)

(* Visualisation DALI_cfg
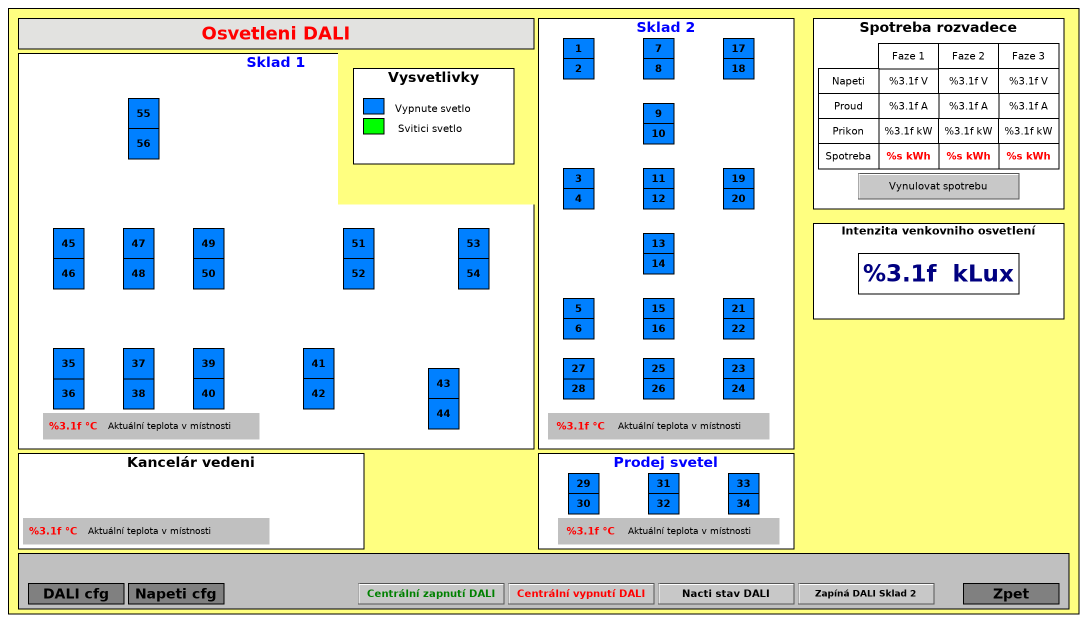
rectangle at (25,55)-(541,451): text "Sklad 1"
rounded rectangle at (360,70)-(521,166): text "Vysvetlivky"
rectangle at (545,455)-(801,551): text "Prodej svetel"; opens prodej_svetel
rectangle at (545,20)-(801,451): text "Sklad 2"; opens prodej_svetel
rectangle at (570,40)-(601,61): text "1"; alarm colour if DALI_Config.Kurzadr[1]
rectangle at (570,40)-(601,61): text "1"; invisible if not DALI_Config.Kurzadr[1]; alarm colour if DALI_Config.LampeEin[1]
rectangle at (570,60)-(601,81): text "2"; alarm colour if DALI_Config.Kurzadr[2]
rectangle at (570,60)-(601,81): text "2"; invisible if not DALI_Config.Kurzadr[2]; alarm colour if DALI_Config.LampeEin[2]
rectangle at (570,170)-(601,191): text "3"; alarm colour if DALI_Config.Kurzadr[3]
rectangle at (570,170)-(601,191): text "3"; invisible if not DALI_Config.Kurzadr[3]; alarm colour if DALI_Config.LampeEin[3]
rectangle at (570,190)-(601,211): text "4"; alarm colour if DALI_Config.Kurzadr[4]
rectangle at (570,190)-(601,211): text "4"; invisible if not DALI_Config.Kurzadr[4]; alarm colour if DALI_Config.LampeEin[4]
rectangle at (570,300)-(601,321): text "5"; alarm colour if DALI_Config.Kurzadr[5]
rectangle at (570,300)-(601,321): text "5"; invisible if not DALI_Config.Kurzadr[5]; alarm colour if DALI_Config.LampeEin[5]
rectangle at (570,320)-(601,341): text "6"; alarm colour if DALI_Config.Kurzadr[6]
rectangle at (570,320)-(601,341): text "6"; invisible if not DALI_Config.Kurzadr[6]; alarm colour if DALI_Config.LampeEin[6]
rectangle at (650,40)-(681,61): text "7"; alarm colour if DALI_Config.Kurzadr[7]
rectangle at (650,40)-(681,61): text "7"; invisible if not DALI_Config.Kurzadr[7]; alarm colour if DALI_Config.LampeEin[7]
rectangle at (650,60)-(681,81): text "8"; alarm colour if DALI_Config.Kurzadr[8]
rectangle at (650,60)-(681,81): text "8"; invisible if not DALI_Config.Kurzadr[8]; alarm colour if DALI_Config.LampeEin[8]
rectangle at (650,105)-(681,126): text "9"; alarm colour if DALI_Config.Kurzadr[9]
rectangle at (650,105)-(681,126): text "9"; invisible if not DALI_Config.Kurzadr[9]; alarm colour if DALI_Config.LampeEin[9]
rectangle at (650,125)-(681,146): text "10"; alarm colour if DALI_Config.Kurzadr[10]
rectangle at (650,125)-(681,146): text "10"; invisible if not DALI_Config.Kurzadr[10]; alarm colour if DALI_Config.LampeEin[10]
rectangle at (650,170)-(681,191): text "11"; alarm colour if DALI_Config.Kurzadr[11]
rectangle at (650,170)-(681,191): text "11"; invisible if not DALI_Config.Kurzadr[11]; alarm colour if DALI_Config.LampeEin[11]
rectangle at (650,190)-(681,211): text "12"; alarm colour if DALI_Config.Kurzadr[12]
rectangle at (650,190)-(681,211): text "12"; invisible if not DALI_Config.Kurzadr[12]; alarm colour if DALI_Config.LampeEin[12]
rectangle at (650,235)-(681,256): text "13"; alarm colour if DALI_Config.Kurzadr[13]
rectangle at (650,235)-(681,256): text "13"; invisible if not DALI_Config.Kurzadr[13]; alarm colour if DALI_Config.LampeEin[13]
rectangle at (650,255)-(681,276): text "14"; alarm colour if DALI_Config.Kurzadr[14]
rectangle at (650,255)-(681,276): text "14"; invisible if not DALI_Config.Kurzadr[14]; alarm colour if DALI_Config.LampeEin[14]
rectangle at (650,300)-(681,321): text "15"; alarm colour if DALI_Config.Kurzadr[15]
rectangle at (650,300)-(681,321): text "15"; invisible if not DALI_Config.Kurzadr[15]; alarm colour if DALI_Config.LampeEin[15]
rectangle at (650,320)-(681,341): text "16"; alarm colour if DALI_Config.Kurzadr[16]
rectangle at (650,320)-(681,341): text "16"; invisible if not DALI_Config.Kurzadr[16]; alarm colour if DALI_Config.LampeEin[16]
rectangle at (730,40)-(761,61): text "17"; alarm colour if DALI_Config.Kurzadr[17]
rectangle at (730,40)-(761,61): text "17"; invisible if not DALI_Config.Kurzadr[17]; alarm colour if DALI_Config.LampeEin[17]
rectangle at (730,170)-(761,191): text "19"; alarm colour if DALI_Config.Kurzadr[19]
rectangle at (730,170)-(761,191): text "19"; invisible if not DALI_Config.Kurzadr[19]; alarm colour if DALI_Config.LampeEin[19]
rectangle at (730,60)-(761,81): text "18"; alarm colour if DALI_Config.Kurzadr[18]
rectangle at (730,60)-(761,81): text "18"; invisible if not DALI_Config.Kurzadr[18]; alarm colour if DALI_Config.LampeEin[18]
rectangle at (730,190)-(761,211): text "20"; alarm colour if DALI_Config.Kurzadr[20]
rectangle at (730,190)-(761,211): text "20"; invisible if not DALI_Config.Kurzadr[20]; alarm colour if DALI_Config.LampeEin[20]
rectangle at (730,300)-(761,321): text "21"; alarm colour if DALI_Config.Kurzadr[21]
rectangle at (730,300)-(761,321): text "21"; invisible if not DALI_Config.Kurzadr[21]; alarm colour if DALI_Config.LampeEin[21]
rectangle at (730,320)-(761,341): text "22"; alarm colour if DALI_Config.Kurzadr[22]
rectangle at (730,320)-(761,341): text "22"; invisible if not DALI_Config.Kurzadr[22]; alarm colour if DALI_Config.LampeEin[22]
rectangle at (730,360)-(761,381): text "23"; alarm colour if DALI_Config.Kurzadr[23]
rectangle at (730,360)-(761,381): text "23"; invisible if not DALI_Config.Kurzadr[23]; alarm colour if DALI_Config.LampeEin[23]
rectangle at (730,380)-(761,401): text "24"; alarm colour if DALI_Config.Kurzadr[24]
rectangle at (730,380)-(761,401): text "24"; invisible if not DALI_Config.Kurzadr[24]; alarm colour if DALI_Config.LampeEin[24]
rectangle at (650,360)-(681,381): text "25"; alarm colour if DALI_Config.Kurzadr[25]
rectangle at (650,360)-(681,381): text "25"; invisible if not DALI_Config.Kurzadr[25]; alarm colour if DALI_Config.LampeEin[25]
rectangle at (575,475)-(606,496): text "29"; alarm colour if DALI_Config.Kurzadr[29]
rectangle at (575,475)-(606,496): text "29"; invisible if not DALI_Config.Kurzadr[29]; alarm colour if DALI_Config.LampeEin[29]
rectangle at (570,380)-(601,401): text "28"; alarm colour if DALI_Config.Kurzadr[28]
rectangle at (570,380)-(601,401): text "28"; invisible if not DALI_Config.Kurzadr[28]; alarm colour if DALI_Config.LampeEin[28]
rectangle at (570,360)-(601,381): text "27"; alarm colour if DALI_Config.Kurzadr[27]
rectangle at (570,360)-(601,381): text "27"; invisible if not DALI_Config.Kurzadr[27]; alarm colour if DALI_Config.LampeEin[27]
rectangle at (650,380)-(681,401): text "26"; alarm colour if DALI_Config.Kurzadr[26]
rectangle at (650,380)-(681,401): text "26"; invisible if not DALI_Config.Kurzadr[26]; alarm colour if DALI_Config.LampeEin[26]
rectangle at (575,495)-(606,516): text "30"; alarm colour if DALI_Config.Kurzadr[30]
rectangle at (575,495)-(606,516): text "30"; invisible if not DALI_Config.Kurzadr[30]; alarm colour if DALI_Config.LampeEin[30]
rectangle at (655,475)-(686,496): text "31"; alarm colour if DALI_Config.Kurzadr[31]
rectangle at (655,475)-(686,496): text "31"; invisible if not DALI_Config.Kurzadr[31]; alarm colour if DALI_Config.LampeEin[31]
rectangle at (655,495)-(686,516): text "32"; alarm colour if DALI_Config.Kurzadr[32]
rectangle at (655,495)-(686,516): text "32"; invisible if not DALI_Config.Kurzadr[32]; alarm colour if DALI_Config.LampeEin[32]
rectangle at (735,475)-(766,496): text "33"; alarm colour if DALI_Config.Kurzadr[33]
rectangle at (735,475)-(766,496): text "33"; invisible if not DALI_Config.Kurzadr[33]; alarm colour if DALI_Config.LampeEin[33]
rectangle at (735,495)-(766,516): text "34"; alarm colour if DALI_Config.Kurzadr[34]
rectangle at (735,495)-(766,516): text "34"; invisible if not DALI_Config.Kurzadr[34]; alarm colour if DALI_Config.LampeEin[34]
rectangle at (60,380)-(91,411): text "36"; alarm colour if DALI_Config.Kurzadr[36]
rectangle at (60,380)-(91,411): text "36"; invisible if not DALI_Config.Kurzadr[36]; alarm colour if DALI_Config.LampeEin[36]
rectangle at (130,380)-(161,411): text "38"; alarm colour if DALI_Config.Kurzadr[38]
rectangle at (130,380)-(161,411): text "38"; invisible if not DALI_Config.Kurzadr[38]; alarm colour if DALI_Config.LampeEin[38]
rectangle at (200,350)-(231,381): text "39"; alarm colour if DALI_Config.Kurzadr[39]
rectangle at (200,350)-(231,381): text "39"; invisible if not DALI_Config.Kurzadr[39]; alarm colour if DALI_Config.LampeEin[39]
rectangle at (130,350)-(161,381): text "37"; alarm colour if DALI_Config.Kurzadr[37]
rectangle at (130,350)-(161,381): text "37"; invisible if not DALI_Config.Kurzadr[37]; alarm colour if DALI_Config.LampeEin[37]
rectangle at (60,350)-(91,381): text "35"; alarm colour if DALI_Config.Kurzadr[35]
rectangle at (60,350)-(91,381): text "35"; invisible if not DALI_Config.Kurzadr[35]; alarm colour if DALI_Config.LampeEin[35]
rectangle at (310,350)-(341,381): text "41"; alarm colour if DALI_Config.Kurzadr[41]
rectangle at (310,350)-(341,381): text "41"; invisible if not DALI_Config.Kurzadr[41]; alarm colour if DALI_Config.LampeEin[41]
rectangle at (310,380)-(341,411): text "42"; alarm colour if DALI_Config.Kurzadr[42]
rectangle at (310,380)-(341,411): text "42"; invisible if not DALI_Config.Kurzadr[42]; alarm colour if DALI_Config.LampeEin[42]
rectangle at (200,380)-(231,411): text "40"; alarm colour if DALI_Config.Kurzadr[40]
rectangle at (200,380)-(231,411): text "40"; invisible if not DALI_Config.Kurzadr[40]; alarm colour if DALI_Config.LampeEin[40]
rectangle at (435,370)-(466,401): text "43"; alarm colour if DALI_Config.Kurzadr[43]
rectangle at (435,370)-(466,401): text "43"; invisible if not DALI_Config.Kurzadr[43]; alarm colour if DALI_Config.LampeEin[43]
rectangle at (435,400)-(466,431): text "44"; alarm colour if DALI_Config.Kurzadr[44]
rectangle at (435,400)-(466,431): text "44"; invisible if not DALI_Config.Kurzadr[44]; alarm colour if DALI_Config.LampeEin[44]
rectangle at (60,230)-(91,261): text "45"; alarm colour if DALI_Config.Kurzadr[45]
rectangle at (60,230)-(91,261): text "45"; invisible if not DALI_Config.Kurzadr[45]; alarm colour if DALI_Config.LampeEin[45]
rectangle at (60,260)-(91,291): text "46"; alarm colour if DALI_Config.Kurzadr[46]
rectangle at (60,260)-(91,291): text "46"; invisible if not DALI_Config.Kurzadr[46]; alarm colour if DALI_Config.LampeEin[46]
rectangle at (130,230)-(161,261): text "47"; alarm colour if DALI_Config.Kurzadr[47]
rectangle at (130,230)-(161,261): text "47"; invisible if not DALI_Config.Kurzadr[47]; alarm colour if DALI_Config.LampeEin[47]
rectangle at (130,260)-(161,291): text "48"; alarm colour if DALI_Config.Kurzadr[48]
rectangle at (130,260)-(161,291): text "48"; invisible if not DALI_Config.Kurzadr[48]; alarm colour if DALI_Config.LampeEin[48]
rectangle at (200,230)-(231,261): text "49"; alarm colour if DALI_Config.Kurzadr[49]
rectangle at (200,230)-(231,261): text "49"; invisible if not DALI_Config.Kurzadr[49]; alarm colour if DALI_Config.LampeEin[49]
rectangle at (200,260)-(231,291): text "50"; alarm colour if DALI_Config.Kurzadr[50]
rectangle at (200,260)-(231,291): text "50"; invisible if not DALI_Config.Kurzadr[50]; alarm colour if DALI_Config.LampeEin[50]
rectangle at (350,230)-(381,261): text "51"; alarm colour if DALI_Config.Kurzadr[51]
rectangle at (350,230)-(381,261): text "51"; invisible if not DALI_Config.Kurzadr[51]; alarm colour if DALI_Config.LampeEin[51]
rectangle at (350,260)-(381,291): text "52"; alarm colour if DALI_Config.Kurzadr[52]
rectangle at (350,260)-(381,291): text "52"; invisible if not DALI_Config.Kurzadr[52]; alarm colour if DALI_Config.LampeEin[52]
rectangle at (465,230)-(496,261): text "53"; alarm colour if DALI_Config.Kurzadr[53]
rectangle at (465,230)-(496,261): text "53"; invisible if not DALI_Config.Kurzadr[53]; alarm colour if DALI_Config.LampeEin[53]
rectangle at (465,260)-(496,291): text "54"; alarm colour if DALI_Config.Kurzadr[54]
rectangle at (465,260)-(496,291): text "54"; invisible if not DALI_Config.Kurzadr[54]; alarm colour if DALI_Config.LampeEin[54]
rectangle at (135,100)-(166,131): text "55"; alarm colour if DALI_Config.Kurzadr[55]
rectangle at (135,100)-(166,131): text "55"; invisible if not DALI_Config.Kurzadr[55]; alarm colour if DALI_Config.LampeEin[55]
rectangle at (135,130)-(166,161): text "56"; alarm colour if DALI_Config.Kurzadr[56]
rectangle at (135,130)-(166,161): text "56"; invisible if not DALI_Config.Kurzadr[56]; alarm colour if DALI_Config.LampeEin[56]
rectangle at (25,20)-(541,51): text "Osvetleni DALI"
button at (665,585)-(801,606): text "Nacti stav DALI"; taps DALI_Config.Status; tooltip Kliknutim nactete status svetel. (sviti, nesviti, vadna).
rectangle at (400,100)-(516,121): text "Vypnute svetlo"
rectangle at (400,120)-(536,141): text "Svitici svetlo"
rectangle at (565,520)-(631,546): text "%3.1f °C"; shows .Teplota_2/10.0
rectangle at (630,520)-(786,546): text "Aktuální teplota v místnosti"
rectangle at (620,415)-(776,441): text "Aktuální teplota v místnosti"
rectangle at (110,415)-(266,441): text "Aktuální teplota v místnosti"
rectangle at (555,415)-(621,441): text "%3.1f °C"; shows .Teplota_1/10.0
rectangle at (50,415)-(111,441): text "%3.1f °C"; shows .Teplota_3/10.0
button at (365,585)-(511,606): text "Centrální zapnutí DALI"; taps DALI_Config.Ein; tooltip Vsechny DALI svetla zapni
button at (515,585)-(661,606): text "Centrální vypnutí DALI"; taps DALI_Config.Aus; tooltip Vsechny DALI svetla vypni
rounded rectangle at (820,20)-(1071,211): text "Spotreba rozvadece"
rectangle at (885,70)-(946,96): text "%3.1f V"; shows TriFaze.arNapeti[1]
rectangle at (885,45)-(946,71): text "Faze 1"
rectangle at (945,45)-(1006,71): text "Faze 2"
rectangle at (1005,45)-(1066,71): text "Faze 3"
rectangle at (945,70)-(1006,96): text "%3.1f V"; shows TriFaze.arNapeti[2]
rectangle at (1005,70)-(1066,96): text "%3.1f V"; shows TriFaze.arNapeti[3]
rectangle at (1005,95)-(1066,121): text "%3.1f A"; shows TriFaze.arProud[3]
rectangle at (945,95)-(1006,121): text "%3.1f A"; shows TriFaze.arProud[2]
rectangle at (885,95)-(946,121): text "%3.1f A"; shows TriFaze.arProud[1]
rectangle at (885,120)-(946,146): text "%3.1f kW"; shows TriFaze.arVykon[1]
rectangle at (945,120)-(1006,146): text "%3.1f kW"; shows TriFaze.arVykon[2]
rectangle at (1005,120)-(1066,146): text "%3.1f kW"; shows TriFaze.arVykon[3]
rectangle at (1005,145)-(1066,171): text "%s kWh"; shows TriFaze.adwSpotreba[3]
rectangle at (945,145)-(1006,171): text "%s kWh"; shows TriFaze.adwSpotreba[2]
rectangle at (885,145)-(946,171): text "%s kWh"; shows TriFaze.adwSpotreba[1]
button at (865,175)-(1026,201): text "Vynulovat spotrebu"; taps TriFaze.SmazL1
rounded rectangle at (820,225)-(1071,321): text "Intenzita venkovniho osvetlení"; opens lux
rectangle at (865,255)-(1026,296): text "%3.1f  kLux"; shows .Analog_1/3276.4*2
rectangle at (825,70)-(886,96): text "Napeti"
rectangle at (825,95)-(886,121): text "Proud"
rectangle at (825,120)-(886,146): text "Prikon"
rectangle at (825,145)-(886,171): text "Spotreba"
rectangle at (25,455)-(371,551): text "Kancelár vedeni"
rectangle at (90,520)-(276,546): text "Aktuální teplota v místnosti"
rectangle at (30,520)-(91,546): text "%3.1f °C"; shows .Teplota_4/10.0
rectangle at (970,585)-(1066,606): text "Zpet"; opens PLC_VISU; tooltip Na úvodní stranu
rectangle at (135,585)-(231,606): text "Napeti cfg"; opens Visualizace; tooltip Back to home page
button at (805,585)-(941,606): text "Zapíná DALI Sklad 2"; taps .TL01s; tooltip 1x zapne/vypne, 2x zapne skupinu 2, 3x zapne vše
rectangle at (35,585)-(131,606): text "DALI cfg"; opens DALI; tooltip Back to home page
6 more shapes without text or variables
*)

(* Visualisation ECG_settings
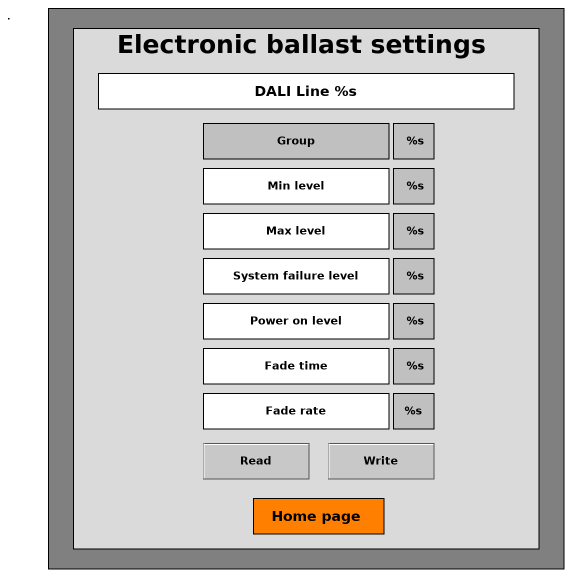
rectangle at (150,40)-(616,561): text "Electronic ballast settings"
rectangle at (280,225)-(466,261): text "Max level"
rectangle at (280,180)-(466,216): text "Min level"
rectangle at (280,270)-(466,306): text "System failure level"
rectangle at (280,315)-(466,351): text "Power on level"
rectangle at (280,360)-(466,396): text "Fade time"
rectangle at (280,405)-(466,441): text "Fade rate"
rectangle at (280,135)-(466,171): text "Short address"; invisible if DALI_Config.Kurzadr_Gruppe; toggles DALI_Config.Kurzadr_Gruppe
rectangle at (280,135)-(466,171): text "Group"; invisible if not DALI_Config.Kurzadr_Gruppe; toggles DALI_Config.Kurzadr_Gruppe; tooltip Selection group or short address
rectangle at (470,135)-(511,171): text "%s"; shows DALI_Config.Adresse; tooltip Enter group (1-16) or short address (1 - 64); editable
rounded rectangle at (330,510)-(461,546): text "Home page"; opens DALI; tooltip Back to home page
rectangle at (470,180)-(511,216): text "%s"; shows DALI_Config.MinLevel; tooltip Minimal brightness level in percent. Min level has to be smaller than max level.; editable
rectangle at (470,225)-(511,261): text "%s"; shows DALI_Config.MaxLevel; tooltip Maximum brightness level in percent; editable
rectangle at (470,270)-(511,306): text "%s"; shows DALI_Config.SystemFailure; tooltip Brightness level in percent in case of a system failure. The value 101 means "MASK".; editable
rectangle at (470,315)-(511,351): text "%s"; shows DALI_Config.PowerOn; tooltip Brightness level in percent if the ECGs are powered on.; editable
rectangle at (470,360)-(511,396): text "%s"; shows DALI_Config.Konfig[4]; tooltip Enter the fade time (0 - 15); editable
rectangle at (470,405)-(511,441): text "%s"; shows DALI_Config.Konfig[5]; tooltip Enter the fade rate (1 -15); editable
button at (280,455)-(386,491): text "Read"; taps DALI_Config.Lese; tooltip If you click the button "Read", the settings of the ECG will be read. Group queries are not possible.
button at (405,455)-(511,491): text "Write"; taps DALI_Config.Schreib; tooltip If you click the button "Write", the new settings will be written into the ECG.
rounded rectangle at (175,85)-(591,121): text "DALI Line %s"; shows DALI_Config.bDali_Linie; tooltip You can change the DALI Line only on the home page.
2 more shapes without text or variables
*)

(* Visualisation Group_assignment
